ADAPTER ITotalReactor (* Adapter Interface *)
  (* Standard: 61499-1 *)
  (* Version 0.0, 11/29/2023, SESA371406, Schneider Electric *)
  PACKAGE SE.Nereda;
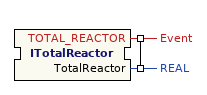
  EVENT_OUTPUT
    TOTAL_REACTOR WITH TotalReactor; (* Confirmation from Plug *)
  END_EVENT
  VAR_OUTPUT
    TotalReactor : REAL; (* Confirmation Data from Plug *)
  END_VAR
  SERVICE SOCKET/PLUG
    SEQUENCE request_confirm
      SOCKET.REQ(REQD) -> PLUG.REQ(REQD);
      PLUG.TOTAL_REACTOR(TotalReactor) -> SOCKET.TOTAL_REACTOR(TotalReactor);
    END_SEQUENCE
    SEQUENCE indication_response
      PLUG.IND(INDD) -> SOCKET.IND(INDD);
      SOCKET.RSP(RSPD) -> PLUG.RSP(RSPD);
    END_SEQUENCE
  END_SERVICE
END_ADAPTER
